{attribute addProperty BoxType "EL2521-0124-0018"}
{attribute addProperty Id "PTO_StatusAT %I*PTO_Status_7C7154A91620ENC_Status_compactAT %I*ENC_Status_compact_EC7EC17A4860PLS_StatusAT %I*PLS_Status_A6235EE11620PTO_ControlAT %Q*PTO_Control_0A6210C33240PTO_Target_compactAT %Q*PTO_Target_compact_C80C22BB1620ENC_Control_compactAT %Q*ENC_Control_compact_5C86AA9D3240PLS_Control_compactAT %Q*PLS_Control_compact_F7E9C6744860WcStateAT %I*WcState_98A4DF7520.250InfoDataAT %I*InfoData_BC63D37F80100"}
{attribute addProperty CRC "2742087237"}
{attribute addProperty SizeInBites "290"}
{attribute addProperty SizeInBytes "36.25"}
TYPE EL2521_880F69EC :
STRUCT
	{attribute addProperty Name "PTO_Status"}
	PTO_Status : PTO_Status_7C7154A9;
	{attribute addProperty Name "ENC_Status_compact"}
	ENC_Status_compact : ENC_Status_compact_EC7EC17A;
	{attribute addProperty Name "PLS_Status"}
	PLS_Status : PLS_Status_A6235EE1;
	{attribute addProperty Name "PTO_Control"}
	PTO_Control : PTO_Control_0A6210C3;
	{attribute addProperty Name "PTO_Target_compact"}
	PTO_Target_compact : PTO_Target_compact_C80C22BB;
	{attribute addProperty Name "ENC_Control_compact"}
	ENC_Control_compact : ENC_Control_compact_5C86AA9D;
	{attribute addProperty Name "PLS_Control_compact"}
	PLS_Control_compact : PLS_Control_compact_F7E9C674;
	{attribute addProperty Name "WcState"}
	WcState : WcState_98A4DF75;
	{attribute addProperty Name "InfoData"}
	InfoData : InfoData_BC63D37F;
END_STRUCT
END_TYPE

(* stored: Version 1.2.0.0, ProductVersion 3.1.4024.9
   DUT EL2521_880F69EC: Id {c8ff5e11-8267-4051-b66b-a088be650310} *)
